// TIA Portal V17 export
// export: Created 2025-03-05T08:02:09.9015955Z, ExportSetting WithDefaults, DisplayName Totally Integrated Automation Portal, DisplayVersion V17 Update 8, DisplayName TIA Portal Openness, DisplayVersion V17 Update 8, DisplayName TIA Portal Version Control Interface, DisplayVersion V17, DisplayName SINAMICS Startdrive Advanced, DisplayVersion V17 SP2, DisplayName SINAMICS Startdrive G110M, G120, G120C, G120D, G120P, G115D, DisplayVersion V17 SP2, DisplayName SINAMICS Startdrive G130, G150, S120, S150, SINAMICS MV, S210, DisplayVersion V17 SP2, DisplayName STEP 7 Professional, DisplayVersion V17 Update 8, DisplayName SINUMERIK ONE STEP 7 Toolbox, DisplayVersion V17 Update 12, DisplayName SINUMERIK 840D sl STEP 7 Toolbox, DisplayVersion V17 Update 12, DisplayName STEP 7 Safety, DisplayVersion V17 Update 6, DisplayName WinCC Advanced, DisplayVersion V17 Update 8
TYPE "CNC_PLC_INT_CH"
// stored: IsFailsafeCompliant false
   STRUCT
      SELECTING_PROG_FAULT_FB : Bool;   // SELECTING PROGRAM FAULT / SELECTING PROGRAM FAULT FB
      SELECTING_PROG_DONE : Bool;   // SELECTING PROGRAM DONE
      REQUEST : Bool;   // REQUEST
      GENERAL_CONDITIONS : Bool;   // GENERAL CONDITIONS
      PULSE : Bool;   // PULSE
      RESET_SELECTION : Bool;   // RESET SELECTION / RESET_SELECTION
      SELECTED : Bool;   // SELECTED
      PROGRAM_SELCT_ALARM : Bool;   // FAULT / PROGRAM SELECTION ALARM
      IS : Bool;   // INMEDIATE STOP ALARMS / IS
      IS_SEOC : Bool;   // INMEDIATE STOP & STOP END OF CYCLE ALARMS / IS_SEOC
      RHP : Bool;   // RETURN HOME POSITION ALARMS / RHP
      RHP_SEOC : Bool;   // RETURN HOME POSITION & STOP END OF CYCLE ALARMS / RHP_SEOC
      SEOC : Bool;   // STOP END OF CYCLE ALARMS / SEOC
      IS_WARNING : Bool;   // INMEDIATE STOP WARNING / IS_WARNING
      RHP_WARNING : Bool;   // RETURN HOME POSITION WARNING / RHP_WARNING
      SEOC_WARNING : Bool;   // STOP END OF CYCLE WARNING / SEOC_WARNING
      WARNINGS : Bool;   // WARNINGS
      HELP : Bool;   // HELP
      Aux : Bool;   // Aux
      Aux1 : Bool;   // Aux1
      Aux2 : Bool;   // Aux2
      Aux3 : Bool;   // Aux3
      Aux4 : Bool;   // Aux4
      Aux5 : Bool;   // Aux5
      Aux6 : Bool;   // Aux6
      Aux7 : Bool;   // Aux7
      SELECTING_STATUS : Word;   // SELECTING STATUS / SELECTING_STATUS
      PName : String[32] := '';   // PName
      Path : String[32] := '';   // Path
   END_STRUCT;
END_TYPE
